// TIA Portal project "iodevice" (V15)

(* hardware
DEVICE "S71500/ET200MP station_1"  S7-1500 station
   slot 0: "Rail_0"  Rack  6ES7 590-1***0-0AA0
   slot 1: "PLC_1"  CPU 1511-1 PN  6ES7 511-1AK00-0AB0  V1.8
      slot 3: "CPU display_1"  6ES7591-1AA00-0AA0
   slot 2: "AI/AQ 4xU/I/RTD/TC / 2xU/I ST_1"  AI/AQ 4xU/I/RTD/TC / 2xU/I ST  6ES7 534-7QE00-0AB0  V1.0
*)

// ===== PLC "PLC_1"  CPU 1511-1 PN =====

VAR_GLOBAL   // PLC tag table "Default tag table"
   "trigger" AT %Q0.0 : Bool;
   "output" AT %Q0.1 : Bool;
   "inturpt" AT %Q0.2 : Bool;
   "genIN" AT %Q0.3 : Bool;
   "genOUT" AT %Q0.4 : Bool;
   "in1" AT %M0.0 : Bool;
   "out1" AT %M0.1 : Bool;
   "out2" AT %M0.2 : Bool;
   "out3" AT %M0.3 : Bool;
   "out3count" AT %MW2 : Int;
   "out1count" AT %MW4 : Int;
   "t1out" AT %M0.4 : Bool;
   "t2out" AT %M0.5 : Bool;
   "t3out" AT %M0.6 : Bool;
   "t4out" AT %M0.7 : Bool;
   "et4" AT %MD6 : Time;
   "et3" AT %MD10 : DWord;
   "et2" AT %MD14 : DWord;
   "et1" AT %MD18 : DInt;
   "timerswitch" AT %M1.0 : Bool;
   "timerswitch(1)" AT %M1.1 : Bool;
   "timerswitch(2)" AT %M1.2 : Bool;
   "timereset" AT %M1.3 : Bool;
   "in2" AT %M1.4 : Bool;
   "reset" AT %M1.5 : Bool;
   "load" AT %M1.6 : Bool;
   "val1" AT %MB22 : USInt;
   "val2" AT %MB23 : USInt;
END_VAR

// folder: System blocks/Program resources

DATA_BLOCK "upcounter"   // DB5
{ S7_Optimized_Access := 'TRUE' }
AUTHOR : Simatic
FAMILY : IEC
NAME : CNTR
VERSION : 1.0
// stored: InstanceOfName IEC_COUNTER
"IEC_COUNTER"
BEGIN
END_DATA_BLOCK

DATA_BLOCK "downcounter"   // DB6
{ S7_Optimized_Access := 'TRUE' }
AUTHOR : Simatic
FAMILY : IEC
NAME : CNTR
VERSION : 1.0
// stored: InstanceOfName IEC_COUNTER
"IEC_COUNTER"
BEGIN
END_DATA_BLOCK

DATA_BLOCK "updown"   // DB7
{ S7_Optimized_Access := 'TRUE' }
AUTHOR : Simatic
FAMILY : IEC
NAME : CNTR
VERSION : 1.0
// stored: InstanceOfName IEC_COUNTER
"IEC_COUNTER"
BEGIN
END_DATA_BLOCK

// folder: (top level)

ORGANIZATION_BLOCK "Main"   // OB1, LAD, ProgramCycle
TITLE = "Main Program Sweep (Cycle)"
{ S7_Optimized_Access := 'TRUE' }
VERSION : 0.1
   VAR_INPUT
      Initial_Call : Bool;   // Initial call of this OB
      Remanence : Bool;   // =True, if remanent data are available
   END_VAR
   VAR_TEMP
      qupdn : Bool;
      qdn : Bool;
      qup : Bool;
      cvupdn : Int;
      cvdn : Int;
      cvup : Int;
      qdupdn : Bool;
   END_VAR
BEGIN

REGION Network 1
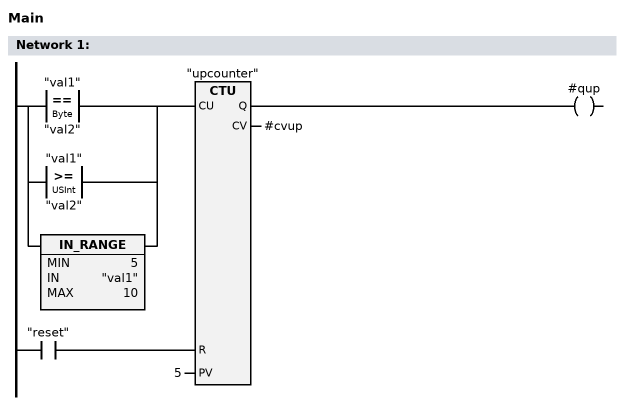
   "upcounter".CTU(CU := ("val1" = "val2") OR ("val1" >= "val2") OR ((5 <= "val1") AND ("val1" <= 10)),
                   R := "reset",
                   PV := 5,
                   CV => #cvup);
   #qup := "upcounter".Q;
END_REGION
END_ORGANIZATION_BLOCK